(* Logix 5000 project; controller Ex_2_05 Emulate 5570 rev 33.11; software revision 33.00 *)
// Turn on lamps with a rotary switch

TASK MainTask (continuous, watchdog 500 ms) : MainProgram

MODULES
   Local : Emulate 5570 (ICP 4, rev 33.11)
END_MODULES

VAR_GLOBAL   (* controller tags *)
   P1 : BOOL;   // Lamp P1
   P2 : BOOL;   // Lamp P2
   S1 : BOOL;   // Rotary Switch S1
END_VAR

PROGRAM MainProgram   (* main routine MainRoutine *)

ROUTINE MainRoutine   (* ladder *)
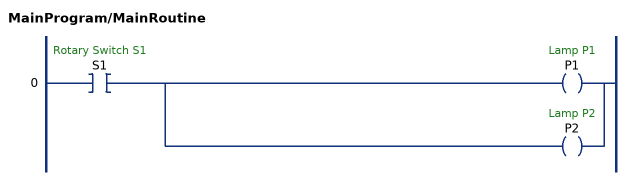
   0: XIC(S1)[OTE(P1) ,OTE(P2) ];
END_ROUTINE
END_PROGRAM
